RoboDK station: Sheet C - Bottom.rdk

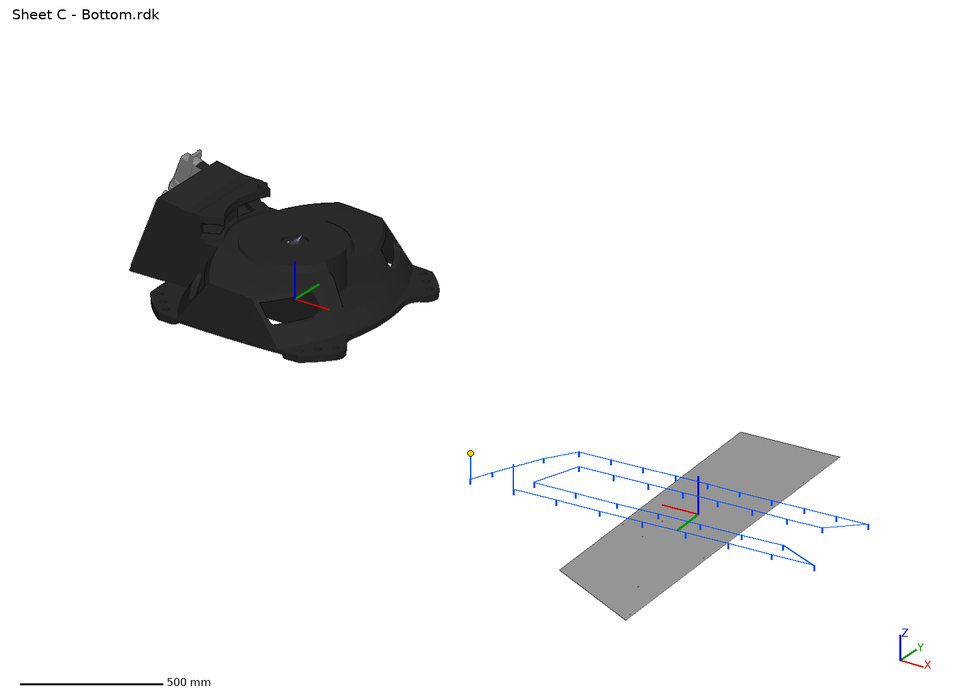
[picture v0: the station drawn from its stored meshes, robots at their saved joint values, targets as dots, program paths as lines]
Station Sheet C - Bottom (saved by RoboDK 5.2.3). Poses are relative to the parent item; angles as X-Y-Z fixed-axis rotations.
  - frame KUKA KR 210 R2700 extra Base at (0, 0, 0) mm
    - robot KUKA KR 210 R2700 extra: 6 axes, payload 210 kg, reach 2696 mm, repeatability 0.06 mm, weight 1068 kg
        joint limits [-185, -140, -120, -350, -125, -350] to [185, -5, 155, 350, 125, 350]; home [0, -90, 90, 0, 0, 0]; saved at [33.004, -28.824, 122.531, -149.283, 42.15, 183.008]
      - tool Spindle, TCP at (32, 0, 260) mm, rotated rx 0 ry 39 rz 0 deg, size 157.3 x 72 x 259.9 mm
  - frame Frame 2 at (1698.49, 32.25, -372.68) mm, rotated rx 0 ry 0 rz -174.91 deg
    - object Box 2 - Sheet C - Bottom at (0, 0, 0) mm, size 400 x 1500 x 0.8 mm, geometry from Box 2 - Sheet C - Bottom.stl
    - object Box 2 - Sheet C -Bottom at (0, 0, 0) mm, rotated rx 0 ry 0 rz 90 deg, 36 curves, geometry from Point 36
  - machining project Point settings: rotZ(0) | rotX(0)*rotY(0) | rotz(0) | onStart | onPathStart | onApproach | onPoint | onRetract | onFinish | SetRPM(%1) | SetTool(%1) | Extruder(%1) | default | default | OutOnMov(%1) | OutOffMov(%1) | onPathFinish | M_RunCode(%1)
  - program Point (191 instructions, listed below)
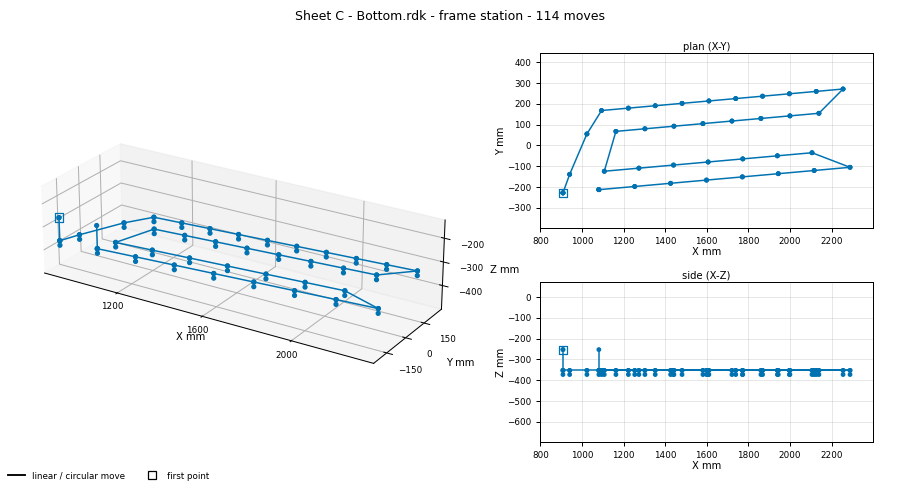
[picture p0: tool path of Sheet C - Bottom.rdk in frame station, 114 of 114 moves have a stored position in this frame; points joined in program order, loops and branches not executed]

--- program Point (robot KUKA KR 210 R2700 extra) ---
  Smooth(1)
  Set speed (1000.0 mm/s)
  Set Ref.: Frame 2
  Set Tool: Spindle
  Show Spindle
  MoveJ 1 to (810.01, 189, 120) mm, rotated rx 180 ry 0 rz -95.09 deg; joints [24.221, -28.984, 92.88, -123.893, 18.121, 144.525]
  MoveL 2 to (810.01, 189, 120) mm, rotated rx 180 ry 0 rz -95.09 deg; joints [24.221, -28.984, 92.88, -123.893, 18.121, 144.525]
  MoveL 3 to (810.01, 189, 20) mm, rotated rx -180 ry 0 rz -95.09 deg; joints [24.221, -24.39, 90.434, -128.982, 19.398, 149.898]
  MoveL 4 to (810.01, 189, 20) mm, rotated rx -180 ry 0 rz -95.09 deg; joints [24.221, -24.39, 90.434, -128.982, 19.398, 149.898]
  Set speed (50.0 mm/s)
  MoveL 5 to (810.01, 189, 0) mm, rotated rx 180 ry 0 rz -95.09 deg; joints [24.221, -23.464, 89.895, -129.826, 19.644, 150.794]
  MoveL 6 to (810.01, 189, 20) mm, rotated rx -180 ry 0 rz -95.09 deg; joints [24.221, -24.39, 90.434, -128.982, 19.398, 149.898]
  Set speed (1000.0 mm/s)
  MoveL 7 to (770, 103, 20) mm, rotated rx -180 ry 0 rz -95.09 deg; joints [24.457, -26.004, 96.149, -136.532, 22.254, 158.205]
  Set speed (50.0 mm/s)
  MoveL 8 to (770, 103, 0) mm, rotated rx 180 ry 0 rz -95.09 deg; joints [24.457, -25.045, 95.606, -137.22, 22.557, 158.95]
  MoveL 9 to (770, 103, 20) mm, rotated rx -180 ry 0 rz -95.09 deg; joints [24.457, -26.004, 96.149, -136.532, 22.254, 158.205]
  Set speed (1000.0 mm/s)
  MoveL 10 to (670.16, -83, 20) mm, rotated rx 180 ry 0 rz -95.09 deg; joints [24.637, -28.493, 107.874, -147.95, 29.629, 171.061]
  Set speed (50.0 mm/s)
  MoveL 11 to (670.16, -83, 0) mm, rotated rx -180 ry 0 rz -95.09 deg; joints [24.637, -27.447, 107.303, -148.387, 30.032, 171.564]
  MoveL 12 to (670.16, -83, 20) mm, rotated rx 180 ry 0 rz -95.09 deg; joints [24.637, -28.493, 107.874, -147.95, 29.629, 171.061]
  Set speed (1000.0 mm/s)
  MoveL 13 to (590.01, -189, 20) mm, rotated rx 180 ry 0 rz -95.09 deg; joints [23.945, -29.198, 114.569, -153.423, 34.813, 176.711]
  Set speed (50.0 mm/s)
  MoveL 14 to (590.01, -189, 0) mm, rotated rx 180 ry 0 rz -95.09 deg; joints [23.945, -28.088, 113.969, -153.747, 35.269, 177.106]
  MoveL 15 to (590.01, -189, 20) mm, rotated rx 180 ry 0 rz -95.09 deg; joints [23.945, -29.198, 114.569, -153.423, 34.813, 176.711]
  Set speed (1000.0 mm/s)
  MoveL 16 to (460.45, -189, 20) mm, rotated rx 180 ry 0 rz -95.09 deg; joints [19.138, -29.272, 117.383, -160.057, 37.22, 178.976]
  Set speed (50.0 mm/s)
  MoveL 17 to (460.45, -189, 0) mm, rotated rx -180 ry 0 rz -95.09 deg; joints [19.138, -28.132, 116.768, -160.289, 37.713, 179.269]
  MoveL 18 to (460.45, -189, 20) mm, rotated rx 180 ry 0 rz -95.09 deg; joints [19.138, -29.272, 117.383, -160.057, 37.22, 178.976]
  Set speed (1000.0 mm/s)
  MoveL 19 to (330.9, -189, 20) mm, rotated rx -180 ry 0 rz -95.09 deg; joints [13.939, -29.213, 119.634, -166.184, 39.408, 180.16]
  Set speed (50.0 mm/s)
  MoveL 20 to (330.9, -189, 0) mm, rotated rx 180 ry 0 rz -95.09 deg; joints [13.939, -28.048, 119.004, -166.337, 39.928, 180.359]
  MoveL 21 to (330.9, -189, 20) mm, rotated rx -180 ry 0 rz -95.09 deg; joints [13.939, -29.213, 119.634, -166.184, 39.408, 180.16]
  Set speed (1000.0 mm/s)
  MoveL 22 to (201.34, -189, 20) mm, rotated rx 180 ry 0 rz -95.09 deg; joints [8.395, -29.091, 121.304, -171.981, 41.191, 180.491]
  Set speed (50.0 mm/s)
  MoveL 23 to (201.34, -189, 0) mm, rotated rx 180 ry 0 rz -95.09 deg; joints [8.395, -27.907, 120.663, -172.066, 41.728, 180.604]
  MoveL 24 to (201.34, -189, 20) mm, rotated rx 180 ry 0 rz -95.09 deg; joints [8.395, -29.091, 121.304, -171.981, 41.191, 180.491]
  Set speed (1000.0 mm/s)
  MoveL 25 to (71.79, -189, 20) mm, rotated rx -180 ry 0 rz -95.09 deg; joints [2.582, -28.972, 122.381, -177.591, 42.406, 180.228]
  Set speed (50.0 mm/s)
  MoveL 26 to (71.79, -189, 0) mm, rotated rx -180 ry 0 rz -95.09 deg; joints [2.582, -27.776, 121.732, -177.616, 42.952, 180.261]
  MoveL 27 to (71.79, -189, 20) mm, rotated rx -180 ry 0 rz -95.09 deg; joints [2.582, -28.972, 122.381, -177.591, 42.406, 180.228]
  Set speed (1000.0 mm/s)
  MoveL 28 to (-57.77, -189, 20) mm, rotated rx 180 ry 0 rz -95.09 deg; joints [-3.395, -28.909, 122.855, -183.136, 42.94, 179.657]
  Set speed (50.0 mm/s)
  MoveL 29 to (-57.77, -189, 0) mm, rotated rx 180 ry 0 rz -95.09 deg; joints [-3.395, -27.707, 122.202, -183.104, 43.488, 179.614]
  MoveL 30 to (-57.77, -189, 20) mm, rotated rx 180 ry 0 rz -95.09 deg; joints [-3.395, -28.909, 122.855, -183.136, 42.94, 179.657]
  Set speed (1000.0 mm/s)
  MoveL 31 to (-187.32, -189, 20) mm, rotated rx 180 ry 0 rz -95.09 deg; joints [-9.408, -28.927, 122.722, -188.717, 42.748, 179.087]
  Set speed (50.0 mm/s)
  MoveL 32 to (-187.32, -189, 0) mm, rotated rx 180 ry 0 rz -95.09 deg; joints [-9.408, -27.727, 122.071, -188.628, 43.29, 178.965]
  MoveL 33 to (-187.32, -189, 20) mm, rotated rx 180 ry 0 rz -95.09 deg; joints [-9.408, -28.927, 122.722, -188.717, 42.748, 179.087]
  Set speed (1000.0 mm/s)
  MoveL 34 to (-316.88, -189, 20) mm, rotated rx -180 ry 0 rz -95.09 deg; joints [-15.328, -29.02, 121.984, -194.434, 41.865, 178.826]
  Set speed (50.0 mm/s)
  MoveL 35 to (-316.88, -189, 0) mm, rotated rx 180 ry 0 rz -95.09 deg; joints [-15.328, -27.828, 121.338, -194.284, 42.394, 178.625]
  MoveL 36 to (-316.88, -189, 20) mm, rotated rx -180 ry 0 rz -95.09 deg; joints [-15.328, -29.02, 121.984, -194.434, 41.865, 178.826]
  Set speed (1000.0 mm/s)
  MoveL 37 to (-446.43, -189, 20) mm, rotated rx 180 ry 0 rz -95.09 deg; joints [-21.035, -29.147, 120.646, -200.396, 40.402, 179.17]
  Set speed (50.0 mm/s)
  MoveL 38 to (-446.43, -189, 0) mm, rotated rx 180 ry 0 rz -95.09 deg; joints [-21.035, -27.971, 120.01, -200.178, 40.908, 178.883]
  MoveL 39 to (-446.43, -189, 20) mm, rotated rx 180 ry 0 rz -95.09 deg; joints [-21.035, -29.147, 120.646, -200.396, 40.402, 179.17]
  Set speed (1000.0 mm/s)
  MoveL 40 to (-575.99, -189, 20) mm, rotated rx 180 ry 0 rz -95.09 deg; joints [-26.436, -29.251, 118.721, -206.731, 38.526, 180.379]
  Set speed (50.0 mm/s)
  MoveL 41 to (-575.99, -189, 0) mm, rotated rx -180 ry 0 rz -95.09 deg; joints [-26.436, -28.096, 118.097, -206.436, 39, 180]
  MoveL 42 to (-575.99, -189, 20) mm, rotated rx 180 ry 0 rz -95.09 deg; joints [-26.436, -29.251, 118.721, -206.731, 38.526, 180.379]
  Set speed (1000.0 mm/s)
  MoveL 43 to (-450, -83, 20) mm, rotated rx 180 ry 0 rz -95.09 deg; joints [-19.972, -29.248, 115.776, -201.585, 35.753, 182.029]
  Set speed (50.0 mm/s)
  MoveL 44 to (-450, -83, 0) mm, rotated rx 180 ry 0 rz -95.09 deg; joints [-19.972, -28.126, 115.17, -201.325, 36.234, 181.708]
  MoveL 45 to (-450, -83, 20) mm, rotated rx 180 ry 0 rz -95.09 deg; joints [-19.972, -29.248, 115.776, -201.585, 35.753, 182.029]
  Set speed (1000.0 mm/s)
  MoveL 46 to (-309.98, -83, 20) mm, rotated rx 180 ry 0 rz -95.09 deg; joints [-14.245, -29.272, 117.182, -194.918, 36.977, 180.855]
  Set speed (50.0 mm/s)
  MoveL 47 to (-309.98, -83, 0) mm, rotated rx 180 ry 0 rz -95.09 deg; joints [-14.245, -28.134, 116.568, -194.742, 37.483, 180.633]
  MoveL 48 to (-309.98, -83, 20) mm, rotated rx 180 ry 0 rz -95.09 deg; joints [-14.245, -29.272, 117.182, -194.918, 36.977, 180.855]
  Set speed (1000.0 mm/s)
  MoveL 49 to (-169.96, -83, 20) mm, rotated rx 180 ry 0 rz -95.09 deg; joints [-8.327, -29.268, 117.902, -188.581, 37.649, 180.324]
  Set speed (50.0 mm/s)
  MoveL 50 to (-169.96, -83, 0) mm, rotated rx 180 ry 0 rz -95.09 deg; joints [-8.327, -28.123, 117.284, -188.481, 38.17, 180.197]
  MoveL 51 to (-169.96, -83, 20) mm, rotated rx 180 ry 0 rz -95.09 deg; joints [-8.327, -29.268, 117.902, -188.581, 37.649, 180.324]
  Set speed (1000.0 mm/s)
  MoveL 52 to (-29.94, -83, 20) mm, rotated rx 180 ry 0 rz -95.09 deg; joints [-2.34, -29.268, 117.93, -182.41, 37.664, 180.089]
  Set speed (50.0 mm/s)
  MoveL 53 to (-29.94, -83, 0) mm, rotated rx 180 ry 0 rz -95.09 deg; joints [-2.34, -28.122, 117.312, -182.381, 38.19, 180.054]
  MoveL 54 to (-29.94, -83, 20) mm, rotated rx 180 ry 0 rz -95.09 deg; joints [-2.34, -29.268, 117.93, -182.41, 37.664, 180.089]
  Set speed (1000.0 mm/s)
  MoveL 55 to (110.08, -83, 20) mm, rotated rx -180 ry 0 rz -95.09 deg; joints [3.588, -29.272, 117.266, -176.247, 36.998, 179.791]
  Set speed (50.0 mm/s)
  MoveL 56 to (110.08, -83, 0) mm, rotated rx -180 ry 0 rz -95.09 deg; joints [3.588, -28.134, 116.652, -176.292, 37.521, 179.848]
  MoveL 57 to (110.08, -83, 20) mm, rotated rx -180 ry 0 rz -95.09 deg; joints [3.588, -29.272, 117.266, -176.247, 36.998, 179.791]
  Set speed (1000.0 mm/s)
  MoveL 58 to (250.1, -83, 20) mm, rotated rx 180 ry 0 rz -95.09 deg; joints [9.336, -29.252, 115.916, -169.927, 35.712, 179.073]
  Set speed (50.0 mm/s)
  MoveL 59 to (250.1, -83, 0) mm, rotated rx -180 ry 0 rz -95.09 deg; joints [9.336, -28.128, 115.309, -170.051, 36.221, 179.226]
  MoveL 60 to (250.1, -83, 20) mm, rotated rx 180 ry 0 rz -95.09 deg; joints [9.336, -29.252, 115.916, -169.927, 35.712, 179.073]
  Set speed (1000.0 mm/s)
  MoveL 61 to (390.12, -83, 20) mm, rotated rx 180 ry 0 rz -95.09 deg; joints [14.802, -29.158, 113.891, -163.26, 33.93, 177.592]
  Set speed (50.0 mm/s)
  MoveL 62 to (390.12, -83, 0) mm, rotated rx -180 ry 0 rz -95.09 deg; joints [14.802, -28.055, 113.294, -163.473, 34.416, 177.85]
  MoveL 63 to (390.12, -83, 20) mm, rotated rx 180 ry 0 rz -95.09 deg; joints [14.802, -29.158, 113.891, -163.26, 33.93, 177.592]
  Set speed (1000.0 mm/s)
  MoveL 64 to (530.14, -83, 20) mm, rotated rx 180 ry 0 rz -95.09 deg; joints [19.916, -28.926, 111.205, -156.019, 31.833, 175.022]
  Set speed (50.0 mm/s)
  MoveL 65 to (530.14, -83, 0) mm, rotated rx 180 ry 0 rz -95.09 deg; joints [19.916, -27.849, 110.621, -156.337, 32.283, 175.397]
  MoveL 66 to (530.14, -83, 20) mm, rotated rx 180 ry 0 rz -95.09 deg; joints [19.916, -28.926, 111.205, -156.019, 31.833, 175.022]
  Set speed (1000.0 mm/s)
  MoveL 67 to (602.86, 103, 20) mm, rotated rx -180 ry 0 rz -95.09 deg; joints [19.481, -27.082, 100.53, -148.856, 23.941, 166.46]
  Set speed (50.0 mm/s)
  MoveL 68 to (602.86, 103, 0) mm, rotated rx 180 ry 0 rz -95.09 deg; joints [19.481, -26.094, 99.979, -149.357, 24.316, 167.009]
  MoveL 69 to (602.86, 103, 20) mm, rotated rx -180 ry 0 rz -95.09 deg; joints [19.481, -27.082, 100.53, -148.856, 23.941, 166.46]
  Set speed (1000.0 mm/s)
  MoveL 70 to (435.71, 103, 20) mm, rotated rx 180 ry 0 rz -95.09 deg; joints [14.077, -27.815, 103.986, -159.388, 25.773, 172.316]
  Set speed (50.0 mm/s)
  MoveL 71 to (435.71, 103, 0) mm, rotated rx -180 ry 0 rz -95.09 deg; joints [14.077, -26.802, 103.427, -159.714, 26.199, 172.678]
  MoveL 72 to (435.71, 103, 20) mm, rotated rx 180 ry 0 rz -95.09 deg; joints [14.077, -27.815, 103.986, -159.388, 25.773, 172.316]
  Set speed (1000.0 mm/s)
  MoveL 73 to (268.57, 103, 20) mm, rotated rx 180 ry 0 rz -95.09 deg; joints [8.296, -28.275, 106.514, -168.623, 27.406, 176.337]
  Set speed (50.0 mm/s)
  MoveL 74 to (268.57, 103, 0) mm, rotated rx -180 ry 0 rz -95.09 deg; joints [8.296, -27.241, 105.948, -168.798, 27.865, 176.534]
  MoveL 75 to (268.57, 103, 20) mm, rotated rx 180 ry 0 rz -95.09 deg; joints [8.296, -28.275, 106.514, -168.623, 27.406, 176.337]
  Set speed (1000.0 mm/s)
  MoveL 76 to (101.43, 103, 20) mm, rotated rx 180 ry 0 rz -95.09 deg; joints [2.224, -28.527, 108.103, -177.075, 28.586, 179.159]
  Set speed (50.0 mm/s)
  MoveL 77 to (101.43, 103, 0) mm, rotated rx 180 ry 0 rz -95.09 deg; joints [2.224, -27.479, 107.531, -177.119, 29.062, 179.209]
  MoveL 78 to (101.43, 103, 20) mm, rotated rx 180 ry 0 rz -95.09 deg; joints [2.224, -28.527, 108.103, -177.075, 28.586, 179.159]
  Set speed (1000.0 mm/s)
  MoveL 79 to (-65.71, 103, 20) mm, rotated rx -180 ry 0 rz -95.09 deg; joints [-4.018, -28.62, 108.743, -185.193, 29.154, 181.414]
  Set speed (50.0 mm/s)
  MoveL 80 to (-65.71, 103, 0) mm, rotated rx -180 ry 0 rz -95.09 deg; joints [-4.018, -27.566, 108.169, -185.116, 29.632, 181.326]
  MoveL 81 to (-65.71, 103, 20) mm, rotated rx -180 ry 0 rz -95.09 deg; joints [-4.018, -28.62, 108.743, -185.193, 29.154, 181.414]
  Set speed (1000.0 mm/s)
  MoveL 82 to (-232.86, 103, 20) mm, rotated rx 180 ry 0 rz -95.09 deg; joints [-10.284, -28.575, 108.428, -193.373, 29.064, 183.712]
  Set speed (50.0 mm/s)
  MoveL 83 to (-232.86, 103, 0) mm, rotated rx 180 ry 0 rz -95.09 deg; joints [-10.284, -27.524, 107.855, -193.177, 29.529, 183.488]
  MoveL 84 to (-232.86, 103, 20) mm, rotated rx 180 ry 0 rz -95.09 deg; joints [-10.284, -28.575, 108.428, -193.373, 29.064, 183.712]
  Set speed (1000.0 mm/s)
  MoveL 85 to (-400, 103, 20) mm, rotated rx 180 ry 0 rz -95.09 deg; joints [-16.429, -28.382, 107.163, -201.985, 28.389, 186.646]
  Set speed (50.0 mm/s)
  MoveL 86 to (-400, 103, 0) mm, rotated rx -180 ry 0 rz -95.09 deg; joints [-16.429, -27.342, 106.594, -201.663, 28.827, 186.28]
  MoveL 87 to (-400, 103, 20) mm, rotated rx 180 ry 0 rz -95.09 deg; joints [-16.429, -28.382, 107.163, -201.985, 28.389, 186.646]
  Set speed (1000.0 mm/s)
  MoveL 88 to (-575.99, 189, 20) mm, rotated rx 180 ry 0 rz -95.09 deg; joints [-21.741, -27.021, 100.264, -214.778, 24.122, 195.148]
  Set speed (50.0 mm/s)
  MoveL 89 to (-575.99, 189, 0) mm, rotated rx -180 ry 0 rz -95.09 deg; joints [-21.741, -26.035, 99.714, -214.232, 24.481, 194.548]
  MoveL 90 to (-575.99, 189, 20) mm, rotated rx 180 ry 0 rz -95.09 deg; joints [-21.741, -27.021, 100.264, -214.778, 24.122, 195.148]
  Set speed (1000.0 mm/s)
  MoveL 91 to (-402.74, 189, 20) mm, rotated rx 180 ry 0 rz -95.09 deg; joints [-15.932, -27.528, 102.569, -204.22, 24.904, 189.687]
  Set speed (50.0 mm/s)
  MoveL 92 to (-402.74, 189, 0) mm, rotated rx -180 ry 0 rz -95.09 deg; joints [-15.932, -26.526, 102.014, -203.831, 25.312, 189.258]
  MoveL 93 to (-402.74, 189, 20) mm, rotated rx 180 ry 0 rz -95.09 deg; joints [-15.932, -27.528, 102.569, -204.22, 24.904, 189.687]
  Set speed (1000.0 mm/s)
  MoveL 94 to (-229.49, 189, 20) mm, rotated rx -180 ry 0 rz -95.09 deg; joints [-9.889, -27.792, 103.866, -194.608, 25.377, 185.534]
  Set speed (50.0 mm/s)
  MoveL 95 to (-229.49, 189, 0) mm, rotated rx -180 ry 0 rz -95.09 deg; joints [-9.889, -26.779, 103.308, -194.37, 25.817, 185.271]
  MoveL 96 to (-229.49, 189, 20) mm, rotated rx -180 ry 0 rz -95.09 deg; joints [-9.889, -27.792, 103.866, -194.608, 25.377, 185.534]
  Set speed (1000.0 mm/s)
  MoveL 97 to (-56.24, 189, 20) mm, rotated rx 180 ry 0 rz -95.09 deg; joints [-3.738, -27.847, 104.151, -185.5, 25.346, 182.067]
  Set speed (50.0 mm/s)
  MoveL 98 to (-56.24, 189, 0) mm, rotated rx -180 ry 0 rz -95.09 deg; joints [-3.738, -26.832, 103.592, -185.409, 25.8, 181.966]
  MoveL 99 to (-56.24, 189, 20) mm, rotated rx 180 ry 0 rz -95.09 deg; joints [-3.738, -27.847, 104.151, -185.5, 25.346, 182.067]
  Set speed (1000.0 mm/s)
  MoveL 100 to (117.01, 189, 20) mm, rotated rx 180 ry 0 rz -95.09 deg; joints [2.383, -27.703, 103.422, -176.416, 24.737, 178.596]
  Set speed (50.0 mm/s)
  MoveL 101 to (117.01, 189, 0) mm, rotated rx 180 ry 0 rz -95.09 deg; joints [2.383, -26.694, 102.864, -176.476, 25.188, 178.662]
  MoveL 102 to (117.01, 189, 20) mm, rotated rx 180 ry 0 rz -95.09 deg; joints [2.383, -27.703, 103.422, -176.416, 24.737, 178.596]
  Set speed (1000.0 mm/s)
  MoveL 103 to (290.26, 189, 20) mm, rotated rx 180 ry 0 rz -95.09 deg; joints [8.337, -27.339, 101.682, -166.826, 23.601, 174.391]
  Set speed (50.0 mm/s)
  MoveL 104 to (290.26, 189, 0) mm, rotated rx 180 ry 0 rz -95.09 deg; joints [8.337, -26.343, 101.129, -167.053, 24.032, 174.639]
  MoveL 105 to (290.26, 189, 20) mm, rotated rx 180 ry 0 rz -95.09 deg; joints [8.337, -27.339, 101.682, -166.826, 23.601, 174.391]
  Set speed (1000.0 mm/s)
  MoveL 106 to (463.51, 189, 20) mm, rotated rx 180 ry 0 rz -95.09 deg; joints [14.011, -26.708, 98.937, -156.128, 22.116, 168.681]
  Set speed (50.0 mm/s)
  MoveL 107 to (463.51, 189, 0) mm, rotated rx 180 ry 0 rz -95.09 deg; joints [14.011, -25.731, 98.39, -156.548, 22.509, 169.135]
  MoveL 108 to (463.51, 189, 20) mm, rotated rx 180 ry 0 rz -95.09 deg; joints [14.011, -26.708, 98.937, -156.128, 22.116, 168.681]
  Set speed (1000.0 mm/s)
  MoveL 109 to (636.76, 189, 20) mm, rotated rx 180 ry 0 rz -95.09 deg; joints [19.321, -25.749, 95.192, -143.673, 20.578, 160.699]
  Set speed (50.0 mm/s)
  MoveL 110 to (636.76, 189, 0) mm, rotated rx 180 ry 0 rz -95.09 deg; joints [19.321, -24.796, 94.65, -144.31, 20.91, 161.38]
  MoveL 111 to (636.76, 189, 20) mm, rotated rx 180 ry 0 rz -95.09 deg; joints [19.321, -25.749, 95.192, -143.673, 20.578, 160.699]
  MoveL 112 to (636.76, 189, 20) mm, rotated rx 180 ry 0 rz -95.09 deg; joints [19.321, -25.749, 95.192, -143.673, 20.578, 160.699]
  Set speed (1000.0 mm/s)
  MoveL 113 to (636.76, 189, 20) mm, rotated rx 180 ry 0 rz -95.09 deg; joints [19.321, -25.749, 95.192, -143.673, 20.578, 160.699]
  MoveL 114 to (636.76, 189, 120) mm, rotated rx -180 ry 0 rz -95.09 deg; joints [19.321, -30.49, 97.66, -139.733, 18.793, 156.515]
